{attribute 'GeneratedUsingTerminal: EL2642-0000-0016'}
{attribute addProperty BoxType "EL2642-0000-0016"}
{attribute addProperty Description "EL2642 2Ch. Multiplexer Ausgang 1x4 Reed-Relais 48V AC/DC, 1A, potential-free"}
{attribute addProperty Physics "KK"}
{attribute addProperty Id "DO_Inputs_DeviceAT %I*DO_Inputs_Device_4A9049C53DO_Group_1_OutputsAT %Q*DO_Group_1_Outputs_59D8C01C4DO_Group_2_OutputsAT %Q*DO_Group_2_Outputs_828082884WcStateAT %I*WcState_9091E0EB2InfoDataAT %I*InfoData_BEF6B88E18"}
{attribute addProperty CRC "3321474279"}
{attribute addProperty Size "31"}
TYPE EL2642_C5F9ACE7 EXTENDS EtcSlaveTerminalBase_947E5A46 :
STRUCT
	{attribute addProperty Name "DO_Inputs_Device"}
	DO_Inputs_Device : DO_Inputs_Device_4A9049C5;
	{attribute addProperty Name "DO_Group_1_Outputs"}
	DO_Group_1_Outputs : DO_Group_1_Outputs_59D8C01C;
	{attribute addProperty Name "DO_Group_2_Outputs"}
	DO_Group_2_Outputs : DO_Group_2_Outputs_82808288;
	{attribute addProperty Name "WcState"}
	WcState : WcState_9091E0EB;
	{attribute addProperty Name "InfoData"}
	InfoData : InfoData_BEF6B88E;
END_STRUCT
END_TYPE

(* stored: Version 1.2.0.0, ProductVersion 3.1.4024.9
   DUT EL2642_C5F9ACE7: Id {7b84e95f-b257-4ecb-b68e-13a8f2580083} *)
